// TIA Portal V19 export
TYPE "Prod_SetUp_Man_Feedbak"
   STRUCT
      Done { ExternalAccessible := 'False'; ExternalVisible := 'False'; ExternalWritable := 'False'} : Bool;
      Done_X : Bool;
      Done_Y : Bool;
      Done_Z : Bool;
      Ack_Eseguito_X { ExternalAccessible := 'False'; ExternalVisible := 'False'; ExternalWritable := 'False'} : Array[1.."SETUP_MAN_OPERATIONS_QTY"] of Bool;
      Ack_Eseguito_Y { ExternalAccessible := 'False'; ExternalVisible := 'False'; ExternalWritable := 'False'} : Array[1.."SETUP_MAN_OP_WITH_CODE_QTY"] of Bool;
   END_STRUCT;
END_TYPE
